INTERFACE I_Task EXTENDS __SYSTEM.IQueryInterface

METHOD Abort
END_METHOD

PROPERTY Available : BOOL
GET
END_GET
END_PROPERTY

PROPERTY Busy : bool
GET
END_GET
END_PROPERTY

METHOD CyclicLogic
END_METHOD

PROPERTY Done : bool
GET
END_GET
END_PROPERTY

PROPERTY Error : bool
GET
END_GET
END_PROPERTY

PROPERTY PUBLIC ErrorId : STRING
GET
END_GET
END_PROPERTY

METHOD PUBLIC Execute : BOOL
END_METHOD

METHOD PUBLIC Free
END_METHOD

PROPERTY Timeout : BOOL
GET
END_GET
END_PROPERTY

END_INTERFACE

(* stored: Version 1.1.0.1
   Itf I_Task: Id {06879b9e-5d97-4d9b-a2dc-57fe5da48e3f}
   Folder Methods: Id {6816a4cb-eea1-4515-ad96-5a64460fa0df}
   Folder Properties: Id {a3467548-07e4-492a-864b-b38e5517bd58}
   Method Abort: Id {21ca12c6-2b9c-4060-a27c-f3cd5549fc6a}
   Property Available: Id {0fdbeec1-cc62-474f-801c-9a69b5c87f9e}
   Get Get: Id {f7f001bb-d9a6-457e-9ea1-d4833d7ea1d7}
   Property Busy: Id {c5019b36-6c55-426c-9c84-8e3e8b521037}
   Get Get: Id {4d1f06e6-0d83-4752-a211-a4ed935d6c49}
   Method CyclicLogic: Id {3fca97f5-ba17-4c76-95d6-f1e6d5092647}
   Property Done: Id {98d98e74-cac1-4684-81cb-bd83702b2ec2}
   Get Get: Id {f8728e1b-c5eb-4849-a6a7-cb5de895e34b}
   Property Error: Id {83c4cfa0-645e-49f4-9f2a-14e4ed9a00e9}
   Get Get: Id {15b59c52-a039-4320-977a-00b361c1a885}
   Property ErrorId: Id {c2c1cc76-1a17-46b4-b4f2-6743ac878248}
   Get Get: Id {a8c7891b-44fd-4b4a-b8c6-a0608791e7d7}
   Method Execute: Id {fdec8d95-194c-4fff-890e-bf447419e9e1}
   Method Free: Id {6e385f10-52e5-47ec-8f30-8406f6d76654}
   Property Timeout: Id {5a3f33bf-b3ba-4f80-9e87-65fd83b38b5e}
   Get Get: Id {766fd1b4-6514-4e9c-8a08-da12c6df0ee4} *)
